FUNCTION_BLOCK FB_SDS
VAR_IN_OUT
    stSDS : ST_SDS;
    stSDSPersistent : ST_SDSPersistent;
END_VAR
VAR
    nIndex: UINT;

    fbStateSetup: FB_StateSetupHelper;
    stDefault: ST_PositionState := (
        fDelta := 0.5,
        fVelocity := 1,
        bMoveOk := TRUE,
        bValid := TRUE
    );
END_VAR


// Check the present homing status
ACT_CheckHomeStatus();

IF NOT stSDSPersistent.bInitialized THEN
    // Do all the required initialization for the persistent data of the sample delivery system.

    stSDSPersistent.stTransferArmSlot.sTag := 'TA';
    stSDSPersistent.stDiffractometerSlot.sTag := 'DF';

    FOR nIndex := E_SDSGarageYStates.T1 to E_SDSGarageYStates.B4 BY 1 DO
        stSDSPersistent.astGarageSlot[nIndex].eState := E_SampleSlotStates.EMPTY;
        stSDSPersistent.astGarageSlot[nIndex].sDesc  := '';
    END_FOR

    stSDSPersistent.astGarageSlot[E_SDSGarageYStates.T1].sTag := 'T1';

    stSDSPersistent.astGarageSlot[E_SDSGarageYStates.T1].fDeg := 0.0;
    stSDSPersistent.astGarageSlot[E_SDSGarageYStates.M1].fDeg := 0.0;
    stSDSPersistent.astGarageSlot[E_SDSGarageYStates.B1].fDeg := 0.0;

    stSDSPersistent.astGarageSlot[E_SDSGarageYStates.T2].fDeg := 90.0;
    stSDSPersistent.astGarageSlot[E_SDSGarageYStates.M2].fDeg := 90.0;
    stSDSPersistent.astGarageSlot[E_SDSGarageYStates.B2].fDeg := 90.0;

    stSDSPersistent.astGarageSlot[E_SDSGarageYStates.T3].fDeg := 180.0;
    stSDSPersistent.astGarageSlot[E_SDSGarageYStates.M3].fDeg := 180.0;
    stSDSPersistent.astGarageSlot[E_SDSGarageYStates.B3].fDeg := 180.0;

    stSDSPersistent.astGarageSlot[E_SDSGarageYStates.T4].fDeg := 270.0;
    stSDSPersistent.astGarageSlot[E_SDSGarageYStates.M4].fDeg := 270.0;
    stSDSPersistent.astGarageSlot[E_SDSGarageYStates.B4].fDeg := 270.0;

    stSDSPersistent.astGarageSlot[E_SDSGarageYStates.T1].fYPos := -100.5;
    stSDSPersistent.astGarageSlot[E_SDSGarageYStates.T2].fYPos := -100.5;
    stSDSPersistent.astGarageSlot[E_SDSGarageYStates.T3].fYPos := -100.5;
    stSDSPersistent.astGarageSlot[E_SDSGarageYStates.T4].fYPos := -100.5;

    stSDSPersistent.astGarageSlot[E_SDSGarageYStates.M1].fYPos := -74.5;
    stSDSPersistent.astGarageSlot[E_SDSGarageYStates.M2].fYPos := -74.5;
    stSDSPersistent.astGarageSlot[E_SDSGarageYStates.M3].fYPos := -74.5;
    stSDSPersistent.astGarageSlot[E_SDSGarageYStates.M4].fYPos := -74.5;

    stSDSPersistent.astGarageSlot[E_SDSGarageYStates.B1].fYPos := -44.5;
    stSDSPersistent.astGarageSlot[E_SDSGarageYStates.B2].fYPos := -44.5;
    stSDSPersistent.astGarageSlot[E_SDSGarageYStates.B3].fYPos := -44.5;
    stSDSPersistent.astGarageSlot[E_SDSGarageYStates.B4].fYPos := -44.5;

    stSDSPersistent.fGarageHeightSafeFromCollision := -40.0;
    stSDSPersistent.fGarageRotationClearanceOffset := 45.0;

    stSDSPersistent.bInitialized := TRUE;
END_IF

IF NOT stSDS.bInitialized THEN
    // Do all the required initialization for the non-persistent data of the sample delivery system.
    stSDS.bHomingRequired := TRUE;

    fbStateSetup(stPositionState:=stDefault, bSetDefault:=TRUE);

    stSDS.bInitialized := TRUE;
END_IF

// Update load/unloadable statuses for the garage, transfer arm, and the diffractometer.
UpdateLoadUnloadAbleStatuses(
    stSDS := stSDS,
    stSDSP := stSDSPersistent
);

// Check if garage is above the threshold to rotate freely without fear of hitting the transfer arm.
ConfirmGarageFreeToRotate(
    stSDS := stSDS,
    stSDSP := stSDSPersistent
);

// Control the sequencing of the sample delivery system.
StateMachine(
    stSDS := stSDS,
    stSDSP := stSDSPersistent
);

// Update the position states
UpdatePositionStates(
    stSDS := stSDS,
    stSDSP := stSDSPersistent
);

// Call state position function blocks.
stSDS.fbTransferArmHPos1D(
    stMotionStage:=stSDS.stTransferArmHStage,
    astPositionState:=stSDS.astTransferArmHPosState,
    eEnumSet:=stSDS.eTransferArmHStateSet,
    eEnumGet:=stSDS.eTransferArmHStateGet,
    bEnable:=TRUE,
    stEpicsToPlc:=stSDS.stTransferArmHEpicsToPlc,
    stPlcToEpics=>stSDS.stTransferArmHPlcToEpics
);
stSDS.fbTransferArmRPos1D(
    stMotionStage:=stSDS.stTransferArmRStage,
    astPositionState:=stSDS.astTransferArmRPosState,
    eEnumSet:=stSDS.eTransferArmRStateSet,
    eEnumGet:=stSDS.eTransferArmRStateGet,
    bEnable:=TRUE,
    stEpicsToPlc:=stSDS.stTransferArmREpicsToPlc,
    stPlcToEpics=>stSDS.stTransferArmRPlcToEpics
);

stSDS.fbGarageYPos1D(
    stMotionStage:=stSDS.stGarageYStage,
    astPositionState:=stSDS.astGarageYPosState,
    eEnumSet:=stSDS.eGarageYStateSet,
    eEnumGet:=stSDS.eGarageYStateGet,
    bEnable:=TRUE,
    stEpicsToPlc:=stSDS.stGarageYEpicsToPlc,
    stPlcToEpics=>stSDS.stGarageYPlcToEpics
);

stSDS.fbGarageRPos1D(
    stMotionStage:=stSDS.stGarageRStage,
    astPositionState:=stSDS.astGarageRPosState,
    eEnumSet:=stSDS.eGarageRStateSet,
    eEnumGet:=stSDS.eGarageRStateGet,
    bEnable:=TRUE,
    stEpicsToPlc:=stSDS.stGarageREpicsToPlc,
    stPlcToEpics=>stSDS.stGarageRPlcToEpics
);

// Ensure UI boolean commands are cleared after holding for one second.
HoldThenClear(b1 := stSDS.stUISelect.bExitManualControl, tHoldDuration := T#1s);
HoldThenClear(b1 := stSDS.stUISelect.bHomeGarage, tHoldDuration := T#1s);
HoldThenClear(b1 := stSDS.stUISelect.bHomeTransferArm, tHoldDuration := T#1s);
HoldThenClear(b1 := stSDS.stUISelect.bLoad, tHoldDuration := T#1s);
HoldThenClear(b1 := stSDS.stUISelect.bLoadArmFromGarage, tHoldDuration := T#1s);
HoldThenClear(b1 := stSDS.stUISelect.bLoadDiffractometerFromArm, tHoldDuration := T#1s);
HoldThenClear(b1 := stSDS.stUISelect.bLoadGarageFromPort, tHoldDuration := T#1s);
HoldThenClear(b1 := stSDS.stUISelect.bLoadUnloadGarageFromPort, tHoldDuration := T#1s);
HoldThenClear(b1 := stSDS.stUISelect.bManualControl, tHoldDuration := T#1s);
HoldThenClear(b1 := stSDS.stUISelect.bProceed, tHoldDuration := T#1s);
HoldThenClear(b1 := stSDS.stUISelect.bUnload, tHoldDuration := T#1s);
HoldThenClear(b1 := stSDS.stUISelect.bUnloadArmToGarage, tHoldDuration := T#1s);
HoldThenClear(b1 := stSDS.stUISelect.bUnloadDiffractometerToArm, tHoldDuration := T#1s);

// Align with the saved selection at the end of each cycle.
stSDS.stUISelect.eGarageSlot := stSDS.eSelectedGarageSlot;

ACTION ACT_CheckHomeStatus:

// ACTION - Check home status

CASE stSDS.nHomingState OF
    0: // Initialization
        stSDS.tonForwardHomingLimit(IN:=FALSE);
        IF stSDS.stTransferArmHStage.nCommand = E_EpicsMotorCmd.HOME AND stSDS.stTransferArmHStage.bBusy THEN
            stSDS.nHomingState := stSDS.nHomingState + 1;
        END_IF
    1: // Homing Sequence Triggered
        stSDS.tonForwardHomingLimit(IN:=stSDS.stTransferArmHStage.Axis.NcToPlc.SetVelo > 0,PT:=T#1s);
        IF stSDS.stTransferArmHStage.nCommand = E_EpicsMotorCmd.HOME AND stSDS.stTransferArmHStage.bHome THEN
            stSDS.nHomingState := stSDS.nHomingState + 1;
            stSDS.tonHomingStateTimeout(IN:=FALSE);
            stSDS.tonForwardHomingLimit(IN:=FALSE);
        ELSIF NOT stSDS.stTransferArmHStage.bBusy THEN
            stSDS.tonHomingStateTimeout(IN:=TRUE,PT:=T#5s);
            stSDS.tonForwardHomingLimit(IN:=FALSE);
            IF stSDS.tonHomingStateTimeout.Q THEN
                stSDS.nHomingState := -1;
            END_IF
        END_IF
    2: // Homing Sequence Successful
        IF F_Limit(stSDS.stTransferArmHStage.stAxisStatus.fActPosition, stSDS.stTransferArmHStage.fHomePosition-0.1, stSDS.stTransferArmHStage.fHomePosition+0.1, TRUE) THEN
            stSDS.bHomingRequired := FALSE;
            stSDS.nHomingState := 0;
            stSDS.tonHomingRequiredTimeout(IN:=FALSE);
            stSDS.tonHomingStateTimeout(IN:=FALSE);
        ELSIF NOT stSDS.stTransferArmHStage.bBusy THEN
            stSDS.tonHomingStateTimeout(IN:=TRUE,PT:=T#5s);
            IF stSDS.tonHomingStateTimeout.Q THEN
                stSDS.nHomingState := -1;
            END_IF
        END_IF
    -1: // Error Handling
        stSDS.nHomingState := 0;
END_CASE

stSDS.tonHomingRequiredTimeout(IN:=NOT stSDS.bHomingRequired,PT:=stSDS.tHomingRequiredTimeoutTime);
IF stSDS.tonHomingRequiredTimeout.Q THEN
    stSDS.bHomingRequired := TRUE;
END_IF
stSDS.fMinUntilHomingRequired := TIME_TO_REAL(stSDS.tonHomingRequiredTimeout.PT - stSDS.tonHomingRequiredTimeout.ET) / 60000;

IF stSDS.stTransferArmHStage.bExecute AND stSDS.bHomingRequired AND stSDS.stTransferArmHStage.fPosition > stSDS.stTransferArmHStage.stAxisStatus.fActPosition AND
    stSDS.stTransferArmHStage.nCommand <> E_EpicsMotorCmd.HOME THEN

    stSDS.stTransferArmHStage.bError := TRUE;
    stSDS.stTransferArmHStage.sCustomErrorMessage := 'Axis homing status overdue. Please home the axis.';
END_IF
END_ACTION


METHOD PRIVATE CheckCanDo2Criteria
VAR_IN_OUT
    bCanDo : BOOL;
    bCantDo : BOOL;
    sErrorMsg : T_MaxString;
END_VAR
VAR_INPUT
    b1 : BOOL;
    b2 : BOOL;
    sErrorMsgTF : T_MaxString;
    sErrorMsgFT : T_MaxString;
    sErrorMsgFF : T_MaxString;
END_VAR

bCanDo := FALSE;

IF b1 AND b2 THEN
    bCanDo := TRUE;
ELSIF b1 AND NOT b2 THEN
    bCantDo := TRUE;
    sErrorMsg := sErrorMsgTF;
ELSIF NOT b1 AND b2 THEN
    bCantDo := TRUE;
    sErrorMsg := sErrorMsgFT ;
ELSE
    bCantDo := TRUE;
    sErrorMsg := sErrorMsgFF;
END_IF
END_METHOD


METHOD PRIVATE CheckCanLoadArmFromGarage
VAR_IN_OUT
    stSDS : ST_SDS;
    stSDSP : ST_SDSPersistent;
END_VAR

stSDS.sStatusMsg := 'Checking if there is an open slot in the transfer arm and at least one full slot in the garage.';

CheckCanDo2Criteria(
    bCanDo := stSDS.bSuccess,
    bCantDo := stSDS.bError,
    sErrorMsg := stSDS.sErrorMsg,
    b1 := stSDS.bGarageUnloadable,
    b2 := stSDS.bTransferArmLoadable,
    sErrorMsgTF := 'The transfer arm is currently full and cannot be used to remove a sample from the garage.',
    sErrorMsgFT := 'The garage is currently empty and therefore no samples can be removed.',
    sErrorMsgFF := 'The garage is currently empty and the transfer arm is full. Therefore, no samples can be removed.'
);
END_METHOD


METHOD PRIVATE CheckCanLoadDiffractometerFromArm
VAR_IN_OUT
    stSDS : ST_SDS;
    stSDSP : ST_SDSPersistent;
END_VAR

stSDS.sStatusMsg := 'Checking if the diffractometer slot is open and if the transfer arm is carrying a sample.';

CheckCanDo2Criteria(
    bCanDo := stSDS.bSuccess,
    bCantDo := stSDS.bError,
    sErrorMsg := stSDS.sErrorMsg,
    b1 := stSDS.bDiffractometerLoadable,
    b2 := stSDS.bTransferArmUnloadable,
    sErrorMsgTF := 'The transfer arm is currently empty and cannot be used to place a sample in the diffractometer.',
    sErrorMsgFT := 'The diffractometer already has a sample in it.',
    sErrorMsgFF := 'The diffractoemter already has a sample and the transfer arm is empty.'
);
END_METHOD


METHOD PRIVATE CheckCanLoadUnloadGarageFromPort
VAR_IN_OUT
    stSDS : ST_SDS;
    stSDSP : ST_SDSPersistent;
END_VAR

stSDS.sStatusMsg := 'Checking if the garage can be loaded or unloaded from the port.';

stSDS.bSuccess := TRUE;
END_METHOD


METHOD PRIVATE CheckCanUnloadArmToGarage
VAR_IN_OUT
    stSDS : ST_SDS;
    stSDSP : ST_SDSPersistent;
END_VAR

stSDS.sStatusMsg := 'Checking if there is an open slot in the garage and if the transfer arm is carrying a sample.';

CheckCanDo2Criteria(
    bCanDo := stSDS.bSuccess,
    bCantDo := stSDS.bError,
    sErrorMsg := stSDS.sErrorMsg,
    b1 := stSDS.bGarageLoadable,
    b2 := stSDS.bTransferArmUnloadable,
    sErrorMsgTF := 'The transfer arm is currently empty and cannot be used to load sample into the garage.',
    sErrorMsgFT := 'The garage is currently full and therefore no samples can be loaded into it.',
    sErrorMsgFF := 'The garage is currently full and the transfer arm is empty.'
);
END_METHOD


METHOD PRIVATE CheckCanUnloadDiffractometerToArm
VAR_IN_OUT
    stSDS : ST_SDS;
    stSDSP : ST_SDSPersistent;
END_VAR

stSDS.sStatusMsg := 'Checking if the diffractometer slot is full and if the transfer arm is empty.';

CheckCanDo2Criteria(
    bCanDo := stSDS.bSuccess,
    bCantDo := stSDS.bError,
    sErrorMsg := stSDS.sErrorMsg,
    b1 := stSDS.bDiffractometerUnloadable,
    b2 := stSDS.bTransferArmLoadable,
    sErrorMsgTF := 'The transfer arm is currently full and cannot be used to unload a sample from the diffractometer.',
    sErrorMsgFT := 'The diffractometer does not have a sample in it.',
    sErrorMsgFF := 'The diffractometeris empty and the transfer arm is full.'
);
END_METHOD


METHOD PRIVATE ConfirmExtraction
VAR_IN_OUT
    stSDS : ST_SDS;
END_VAR

stSDS.bSuccess := FALSE;

stSDS.sStatusMsg := 'Moving transfer arm back a few mm. Please confirm the sample is held by the arm and then click "proceed". If the sample is still in the holder, click "retry" to go back to fine adjustment.';

SetPositionStateWaitForArrivalQuitIfError(
    eStateGet := stSDS.eTransferArmHStateGet,
    stMotionStage := stSDS.stTransferArmHStage,
    eStateSet := stSDS.eTransferArmHStateSet,
    eEnumSet := E_SDSTransferArmHStates.CONFIRM_GARAGE_EXTRACTION,
    bError := stSDS.bError,
    sErrorMsg := stSDS.sErrorMsg,
    bArrived => stSDS.bSuccess
);
END_METHOD


METHOD PRIVATE ConfirmGarageFreeToRotate
VAR_IN_OUT
    stSDS : ST_SDS;
    stSDSP : ST_SDSPersistent;
END_VAR

stSDS.bGarageAboveCollisionHeight := stSDS.stGarageYStage.Axis.NcToPlc.ActPos <= stSDSP.fGarageHeightSafeFromCollision;
END_METHOD


METHOD PRIVATE ConfirmInsertion
VAR_IN_OUT
    stSDS : ST_SDS;
END_VAR

stSDS.bSuccess := FALSE;

stSDS.sStatusMsg := 'Moving transfer arm back a few mm. Please confirm the sample is held by the garage and then click "proceed". If the sample is still in the transfer arm, click "retry" to go back to fine adjustment.';

SetPositionStateWaitForArrivalQuitIfError(
    eStateGet := stSDS.eTransferArmHStateGet,
    stMotionStage := stSDS.stTransferArmHStage,
    eStateSet := stSDS.eTransferArmHStateSet,
    eEnumSet := E_SDSTransferArmHStates.CONFIRM_GARAGE_INSERTION,
    bError := stSDS.bError,
    sErrorMsg := stSDS.sErrorMsg,
    bArrived => stSDS.bSuccess
);
END_METHOD


METHOD PRIVATE ConfirmSampleLoaded
VAR_INPUT
END_VAR
END_METHOD


METHOD PRIVATE ConfirmSampleUnloaded
VAR_INPUT
END_VAR
END_METHOD


METHOD PRIVATE ExtendPrerotateTransferArmForExtraction
VAR_IN_OUT
    stSDS : ST_SDS;
END_VAR
VAR
    bHArrived : BOOL;
    bRArrived : BOOL;
END_VAR

stSDS.bSuccess := FALSE;

stSDS.sStatusMsg := 'Moving transfer arm to nominal sample extraction position and pre-rotating to allow full rotation for unscrewing sample.';

SetPositionStateWaitForArrivalQuitIfError(
    eStateGet := stSDS.eTransferArmHStateGet,
    stMotionStage := stSDS.stTransferArmHStage,
    eStateSet := stSDS.eTransferArmHStateSet,
    eEnumSet := E_SDSTransferArmHStates.GARAGE_SAMPLE_REMOVAL,
    bError := stSDS.bError,
    sErrorMsg := stSDS.sErrorMsg,
    bArrived => bHArrived
);

SetPositionStateWaitForArrivalQuitIfError(
    eStateGet := stSDS.eTransferArmRStateGet,
    stMotionStage := stSDS.stTransferArmRStage,
    eStateSet := stSDS.eTransferArmRStateSet,
    eEnumSet := E_SDSTransferArmRStates.PREROTATE_SAMPLE_REMOVAL,
    bError := stSDS.bError,
    sErrorMsg := stSDS.sErrorMsg,
    bArrived => bRArrived
);

IF bHArrived AND bRArrived THEN
    stSDS.bSuccess := TRUE;
END_IF
END_METHOD


METHOD PRIVATE ExtendPrerotateTransferArmForLoading
VAR_IN_OUT
    stSDS : ST_SDS;
END_VAR
VAR
    bHArrived : BOOL;
    bRArrived : BOOL;
END_VAR

stSDS.bSuccess := FALSE;

stSDS.sStatusMsg := 'Moving transfer arm to nominal sample loading position and pre-rotating to allow full rotation for screwing in sample.';

SetPositionStateWaitForArrivalQuitIfError(
    eStateGet := stSDS.eTransferArmHStateGet,
    stMotionStage := stSDS.stTransferArmHStage,
    eStateSet := stSDS.eTransferArmHStateSet,
    eEnumSet := E_SDSTransferArmHStates.GARAGE_SAMPLE_INSERTION,
    bError := stSDS.bError,
    sErrorMsg := stSDS.sErrorMsg,
    bArrived => bHArrived
);

SetPositionStateWaitForArrivalQuitIfError(
    eStateGet := stSDS.eTransferArmRStateGet,
    stMotionStage := stSDS.stTransferArmRStage,
    eStateSet := stSDS.eTransferArmRStateSet,
    eEnumSet := E_SDSTransferArmRStates.PREROTATE_SAMPLE_INSERTION,
    bError := stSDS.bError,
    sErrorMsg := stSDS.sErrorMsg,
    bArrived => bRArrived
);

IF bHArrived AND bRArrived THEN
    stSDS.bSuccess := TRUE;
END_IF
END_METHOD


METHOD PRIVATE FineAdjustment
VAR_INPUT
END_VAR

stSDS.sStatusMsg := 'Use the individual motor control to do fine adjustment. Click "proceed" to move to the next step.';
END_METHOD


METHOD PRIVATE HoldThenClear
VAR_IN_OUT
    b1 : BOOL;
END_VAR
VAR_INPUT
    tHoldDuration : TIME := T#1s;
END_VAR
VAR_INST
    tonHoldTimer : TON;
END_VAR

tonHoldTimer(IN := b1, PT := tHoldDuration);

IF tonHoldTimer.Q THEN
    b1 := FALSE;
END_IF
END_METHOD


METHOD PRIVATE HomeGarage
VAR_INPUT
    stSDS : ST_SDS;
END_VAR

stSDS.bSuccess := FALSE;

stSDS.sStatusMsg := 'Homing the garage.';

IF stSDS.stGarageRStage.bError THEN
    stSDS.bError := TRUE;
    stSDS.sErrorMsg := 'Garage rotational stage has an active error. Aborting sequence.';
END_IF

HomeStateMachine(
    eHomingState := stSDS.eGarageRHomingState,
    stMotionStage := stSDS.stGarageRStage,
    bError => stSDS.bError,
    sErrorMsg => stSDS.sErrorMsg
);

IF stSDS.eGarageRHomingState = E_SDSHomingState.HOMED THEN
    stSDS.bSuccess := TRUE;
END_IF
END_METHOD


METHOD PRIVATE HomeStateMachine
VAR_IN_OUT
    eHomingState : E_SDSHomingState;
    stMotionStage : ST_MotionStage;
END_VAR
VAR_OUTPUT
    bError : BOOL;
    sErrorMsg : T_MaxString;
END_VAR

CASE eHomingState OF
    E_SDSHomingState.INIT:
        eHomingState := E_SDSHomingState.WAIT_NOT_BUSY;
    E_SDSHomingState.WAIT_NOT_BUSY:
        IF NOT stMotionStage.bBusy THEN
            eHomingState := E_SDSHomingState.TRIGGER_HOMING;
        END_IF
    E_SDSHomingState.TRIGGER_HOMING:
        stMotionStage.bHomeCmd := TRUE;
        IF stMotionStage.nCommand = E_EpicsMotorCmd.HOME AND stMotionStage.bBusy THEN
            eHomingState := E_SDSHomingState.WAIT_FOR_HOMED;
        END_IF
    E_SDSHomingState.WAIT_FOR_HOMED:
        IF stMotionStage.bDone THEN
            eHomingState := E_SDSHomingState.HOMED;
        END_IF
ELSE
    bError := TRUE;
    sErrorMsg := 'Homing sequence triggered an unknown state. Aborting sequence.';
END_CASE
END_METHOD


METHOD PRIVATE HomeTransferArm
VAR_IN_OUT
    stSDS : ST_SDS;
END_VAR

stSDS.bSuccess := FALSE;

stSDS.sStatusMsg := 'Homing the transfer arm.';

IF stSDS.stTransferArmHStage.bError THEN
    stSDS.bError := TRUE;
    stSDS.sErrorMsg := 'Transfer arm horizontal stage has an active error. Aborting sequence.';
END_IF

IF stSDS.stTransferArmRStage.bError THEN
    stSDS.bError := TRUE;
    stSDS.sErrorMsg := 'Transfer arm rotational stage has an active error. Aborting sequence.';
END_IF

HomeStateMachine(
    eHomingState := stSDS.eTransferArmHHomingState,
    stMotionStage := stSDS.stTransferArmHStage,
    bError => stSDS.bError,
    sErrorMsg => stSDS.sErrorMsg
);

HomeStateMachine(
    eHomingState := stSDS.eTransferArmRHomingState,
    stMotionStage := stSDS.stTransferArmRStage,
    bError => stSDS.bError,
    sErrorMsg => stSDS.sErrorMsg
);

IF stSDS.eTransferArmHHomingState = E_SDSHomingState.HOMED AND
   stSDS.eTransferArmRHomingState = E_SDSHomingState.HOMED THEN
    stSDS.bSuccess := TRUE;
END_IF
END_METHOD


METHOD PRIVATE InitHomeGarage
VAR_IN_OUT
    stSDS : ST_SDS;
END_VAR

stSDS.eGarageRHomingState := E_SDSHomingState.INIT;
END_METHOD


METHOD PRIVATE InitHomeTransferArm
VAR_IN_OUT
    stSDS : ST_SDS;
END_VAR

stSDS.eTransferArmHHomingState := E_SDSHomingState.INIT;
stSDS.eTransferArmRHomingState := E_SDSHomingState.INIT;
END_METHOD


METHOD PRIVATE InitRotateGarageForClearance
VAR_IN_OUT
    stSDS : ST_SDS;
    stSDSP : ST_SDSPersistent;
END_VAR

stSDS.fGarageRotationClearancePos := stSDS.stGarageRStage.Axis.NcToPlc.ActPos + stSDSP.fGarageRotationClearanceOffset;
END_METHOD


METHOD PRIVATE InitSelectGarageSlotForLoading
VAR_IN_OUT
    stSDS : ST_SDS;
    stSDSP : ST_SDSPersistent;
END_VAR

FOR nIndex := E_SDSGarageYStates.T1 TO E_SDSGarageYStates.B4 BY 1 DO
    CASE stSDSP.astGarageSlot[nIndex].eState OF
        E_SampleSlotStates.EMPTY:
            stSDS.eSelectedGarageSlot := nIndex;
    END_CASE
END_FOR

IF nIndex > E_SDSGarageYStates.B4 THEN
    stSDS.bError := TRUE;
    stSDS.sErrorMsg := 'There are no empty slots in the garage to load a sample to.';
END_IF
END_METHOD


METHOD PRIVATE InitSelectGarageSlotForRemoval
VAR_IN_OUT
    stSDS : ST_SDS;
    stSDSP : ST_SDSPersistent;
END_VAR

FOR nIndex := E_SDSGarageYStates.T1 TO E_SDSGarageYStates.B4 BY 1 DO
    CASE stSDSP.astGarageSlot[nIndex].eState OF
        E_SampleSlotStates.FULL:
            stSDS.eSelectedGarageSlot := nIndex;
    END_CASE
END_FOR

IF nIndex > E_SDSGarageYStates.B4 THEN
    stSDS.bError := TRUE;
    stSDS.sErrorMsg := 'There are no full slots in the garage to extract a sample from.';
END_IF
END_METHOD


METHOD PRIVATE ManualControl
VAR_INPUT
    stSDS : ST_SDS;
END_VAR
END_METHOD


METHOD PRIVATE MoveToGarageSlotFaceTransferArm
VAR_IN_OUT
    stSDS : ST_SDS;
END_VAR
VAR
    bYArrived : BOOL;
    bRArrived : BOOL;
END_VAR

stSDS.bSuccess := FALSE;

stSDS.sStatusMsg := 'Moving garage to selected slot and facing it towards transfer arm.';

stSDS.eFaceState := E_SDSFaceState.FACE_TRANSFER_ARM;

SetPositionStateWaitForArrivalQuitIfError(
    eStateGet := stSDS.eGarageYStateGet,
    stMotionStage := stSDS.stGarageYStage,
    eStateSet := stSDS.eGarageYStateSet,
    eEnumSet := stSDS.eSelectedGarageSlot,
    bError := stSDS.bError,
    sErrorMsg := stSDS.sErrorMsg,
    bArrived => bYArrived
);

SetPositionStateWaitForArrivalQuitIfError(
    eStateGet := stSDS.eGarageRStateGet,
    stMotionStage := stSDS.stGarageRStage,
    eStateSet := stSDS.eGarageRStateSet,
    eEnumSet := stSDS.eSelectedGarageSlot,
    bError := stSDS.bError,
    sErrorMsg := stSDS.sErrorMsg,
    bArrived => bRArrived
);

IF bYArrived AND bRArrived THEN
    stSDS.bSuccess := TRUE;
END_IF
END_METHOD


METHOD PRIVATE MoveToGarageSlotHeight
VAR_IN_OUT
    stSDS : ST_SDS;
END_VAR

stSDS.bSuccess := FALSE;

stSDS.sStatusMsg := 'Moving garage to selected slot height.';

SetPositionStateWaitForArrivalQuitIfError(
    eStateGet := stSDS.eGarageYStateGet,
    stMotionStage := stSDS.stGarageYStage,
    eStateSet := stSDS.eGarageYStateSet,
    eEnumSet := stSDS.eSelectedGarageSlot,
    bError := stSDS.bError,
    sErrorMsg := stSDS.sErrorMsg,
    bArrived => stSDS.bSuccess
);
END_METHOD


METHOD PRIVATE RetractGarage
VAR_IN_OUT
    stSDS : ST_SDS;
END_VAR

stSDS.bSuccess := FALSE;

stSDS.sStatusMsg := 'Retracting garage.';

SetPositionStateWaitForArrivalQuitIfError(
    eStateGet := stSDS.eGarageYStateGet,
    stMotionStage := stSDS.stGarageYStage,
    eStateSet := stSDS.eGarageYStateSet,
    eEnumSet := E_SDSGarageYStates.RETRACTED,
    bError := stSDS.bError,
    sErrorMsg := stSDS.sErrorMsg,
    bArrived => stSDS.bSuccess
);
END_METHOD


METHOD PRIVATE RotateGarageForClearance
VAR_IN_OUT
    stSDS : ST_SDS;
END_VAR

stSDS.bSuccess := FALSE;

stSDS.sStatusMsg := 'Rotating garage to prevent a collision with the transfer arm sample during movement of the garage.';

IF F_Limit(
       fVal := stSDS.stGarageRStage.Axis.NcToPlc.ActPos,
       fLLim := stSDS.fGarageRotationClearancePos - stSDS.stGarageRStage.stAxisParameters.fTargetPosControlRange,
       fHLim := stSDS.fGarageRotationClearancePos + stSDS.stGarageRStage.stAxisParameters.fTargetPosControlRange,
       bInclusive := FALSE
   ) AND NOT stSDS.stGarageRStage.bBusy THEN
   stSDS.bSuccess := TRUE;
ELSE
    stSDS.stGarageRStage.fPosition := stSDS.fGarageRotationClearancePos;
    stSDS.stGarageRStage.fVelocity := stSDS.fGarageRotationSpeed;
    stSDS.stGarageRStage.bMoveCmd := TRUE;
END_IF
END_METHOD


METHOD PRIVATE RotateGarageForClearanceManual
VAR_IN_OUT
    stSDS : ST_SDS;
END_VAR

stSDS.sStatusMsg := 'Please manually rotate the garage to 45 degrees, to prevent it from colliding with the sample on the transfer arm when raising it up. Click "proceed" when complete.';
END_METHOD


METHOD PRIVATE RotateToFacePort
VAR_IN_OUT
    stSDS : ST_SDS;
END_VAR

stSDS.bSuccess := FALSE;

stSDS.sStatusMsg := 'Rotating garage so that the selected slot faces the side port.';

stSDS.eFaceState := E_SDSFaceState.FACE_SIDE_PORT;

SetPositionStateWaitForArrivalQuitIfError(
    eStateGet := stSDS.eGarageRStateGet,
    stMotionStage := stSDS.stGarageRStage,
    eStateSet := stSDS.eGarageRStateSet,
    eEnumSet := stSDS.eSelectedGarageSlot,
    bError := stSDS.bError,
    sErrorMsg := stSDS.sErrorMsg,
    bArrived => stSDS.bSuccess
);
END_METHOD


METHOD PRIVATE RotateToFaceTransferArm
VAR_IN_OUT
    stSDS : ST_SDS;
END_VAR

stSDS.bSuccess := FALSE;

stSDS.sStatusMsg := 'Rotating garage so that the selected slot faces the transfer arm.';

stSDS.eFaceState := E_SDSFaceState.FACE_TRANSFER_ARM;

SetPositionStateWaitForArrivalQuitIfError(
    eStateGet := stSDS.eGarageRStateGet,
    stMotionStage := stSDS.stGarageRStage,
    eStateSet := stSDS.eGarageRStateSet,
    eEnumSet := stSDS.eSelectedGarageSlot,
    bError := stSDS.bError,
    sErrorMsg := stSDS.sErrorMsg,
    bArrived => stSDS.bSuccess
);
END_METHOD


METHOD PRIVATE ScrewSampleIntoGarage
VAR_IN_OUT
    stSDS : ST_SDS;
END_VAR

stSDS.bSuccess := FALSE;

stSDS.sStatusMsg := 'Screwing sample into garage. Click "proceed" when complete. To go back and retry fine adjustment, click "retry".';

SetPositionStateWaitForArrivalQuitIfError(
    eStateGet := stSDS.eTransferArmRStateGet,
    stMotionStage := stSDS.stTransferArmRStage,
    eStateSet := stSDS.eTransferArmRStateSet,
    eEnumSet := E_SDSTransferArmRStates.SCREW_INTO_GARAGE,
    bError := stSDS.bError,
    sErrorMsg := stSDS.sErrorMsg,
    bArrived => stSDS.bSuccess
);
END_METHOD


METHOD PRIVATE SelectDesiredAction
VAR_INPUT
    stSDS : ST_SDS;
END_VAR

stSDS.sStatusMsg := 'Please select the desired action.';
END_METHOD


METHOD PRIVATE SelectGarageSlotForLoading
VAR_IN_OUT
    stSDS : ST_SDS;
    stSDSP : ST_SDSPersistent;
END_VAR

stSDS.sStatusMsg := 'Please select a valid garage slot to load a sample to and then click "proceed".';

IF stSDS.stUISelect.eGarageSlot >= E_SDSGarageYStates.T1 AND stSDS.stUISelect.eGarageSlot <= E_SDSGarageYStates.B4 THEN
    CASE stSDSP.astGarageSlot[stSDS.stUISelect.eGarageSlot].eState OF
        E_SampleSlotStates.DISABLED:
            stSDS.sErrorMsg := 'The selected garage slot is currently disabled.';
        E_SampleSlotStates.EMPTY:
            stSDS.eSelectedGarageSlot := stSDS.stUISelect.eGarageSlot;
        E_SampleSlotStates.FULL:
            stSDS.sErrorMsg := 'The selected garage slot is currently full.';
    END_CASE
ELSE
    stSDS.sErrorMsg := 'Please select a valid slot from T1 to B4.';
END_IF
END_METHOD


METHOD PRIVATE SelectGarageSlotForRemoval
VAR_IN_OUT
    stSDS : ST_SDS;
    stSDSP : ST_SDSPersistent;
END_VAR

stSDS.sStatusMsg := 'Please select a valid garage slot to retrieve a sample from and then click "proceed".';

IF stSDS.stUISelect.eGarageSlot >= E_SDSGarageYStates.T1 AND stSDS.stUISelect.eGarageSlot <= E_SDSGarageYStates.B4 THEN
    CASE stSDSP.astGarageSlot[stSDS.stUISelect.eGarageSlot].eState OF
        E_SampleSlotStates.DISABLED:
            stSDS.sErrorMsg := 'The selected garage slot is currently disabled.';
        E_SampleSlotStates.EMPTY:
            stSDS.sErrorMsg := 'The selected garage slot is currently empty.';
        E_SampleSlotStates.FULL:
            stSDS.eSelectedGarageSlot := stSDS.stUISelect.eGarageSlot;
    END_CASE
ELSE
    stSDS.sErrorMsg := 'Please select a valid slot from T1 to B4.';
END_IF
END_METHOD


METHOD PRIVATE SelectLoadUnloadGarage
VAR_IN_OUT
    stSDS : ST_SDS;
END_VAR

stSDS.sStatusMsg := 'Select whether you would like to load a sample to the garage or remove a sample to the garage.';

stSDS.bLoadingSelected := FALSE;
stSDS.bUnloadingSelected := FALSE;

IF stSDS.stUISelect.bLoad THEN
    stSDS.bLoadingSelected := TRUE;
ELSIF stSDS.stUISelect.bUnload THEN
    stSDS.bUnloadingSelected := TRUE;
END_IF
END_METHOD


METHOD PRIVATE SetPositionStateWaitForArrivalQuitIfError
VAR_IN_OUT
    eStateGet : UINT;
    stMotionStage : ST_MotionStage;
    eStateSet : UINT;
    bError : BOOL;
    sErrorMsg : T_MaxString;
END_VAR
VAR_INPUT
    eEnumSet : UINT;
END_VAR
VAR_OUTPUT
    bArrived : BOOL;
END_VAR

IF eStateGet = eEnumSet AND
    NOT stMotionStage.bBusy THEN
    bArrived := TRUE;
ELSIF stMotionStage.bError THEN
    bError := TRUE;
    sErrorMsg := 'And axis error occurred. Aborting sequence.';
END_IF

IF eStateGet <> eEnumSet THEN
    eStateSet := eEnumSet;
END_IF
END_METHOD


METHOD PRIVATE SetSeqState
VAR_INPUT
    stSDS : ST_SDS;
    eSeqState : E_SDSState;
END_VAR

stSDS.eSeqState := eSeqState;
END_METHOD


METHOD PRIVATE SetState
VAR_INPUT
    stSDS : ST_SDS;
    eState : E_SDSState;
END_VAR

stSDS.eState := eState;
END_METHOD


METHOD PRIVATE SetSubstate
VAR_INPUT
    stSDS : ST_SDS;
    eSubState : E_SDSState;
END_VAR

stSDS.eSubState := eSubState;
END_METHOD


METHOD PRIVATE StateMachine
VAR_IN_OUT
    stSDS : ST_SDS;
    stSDSP : ST_SDSPersistent;
END_VAR
END_METHOD


METHOD PRIVATE StateMachine_statechart
VAR_IN_OUT
    stSDS : ST_SDS;
    stSDSP : ST_SDSPersistent;
END_VAR
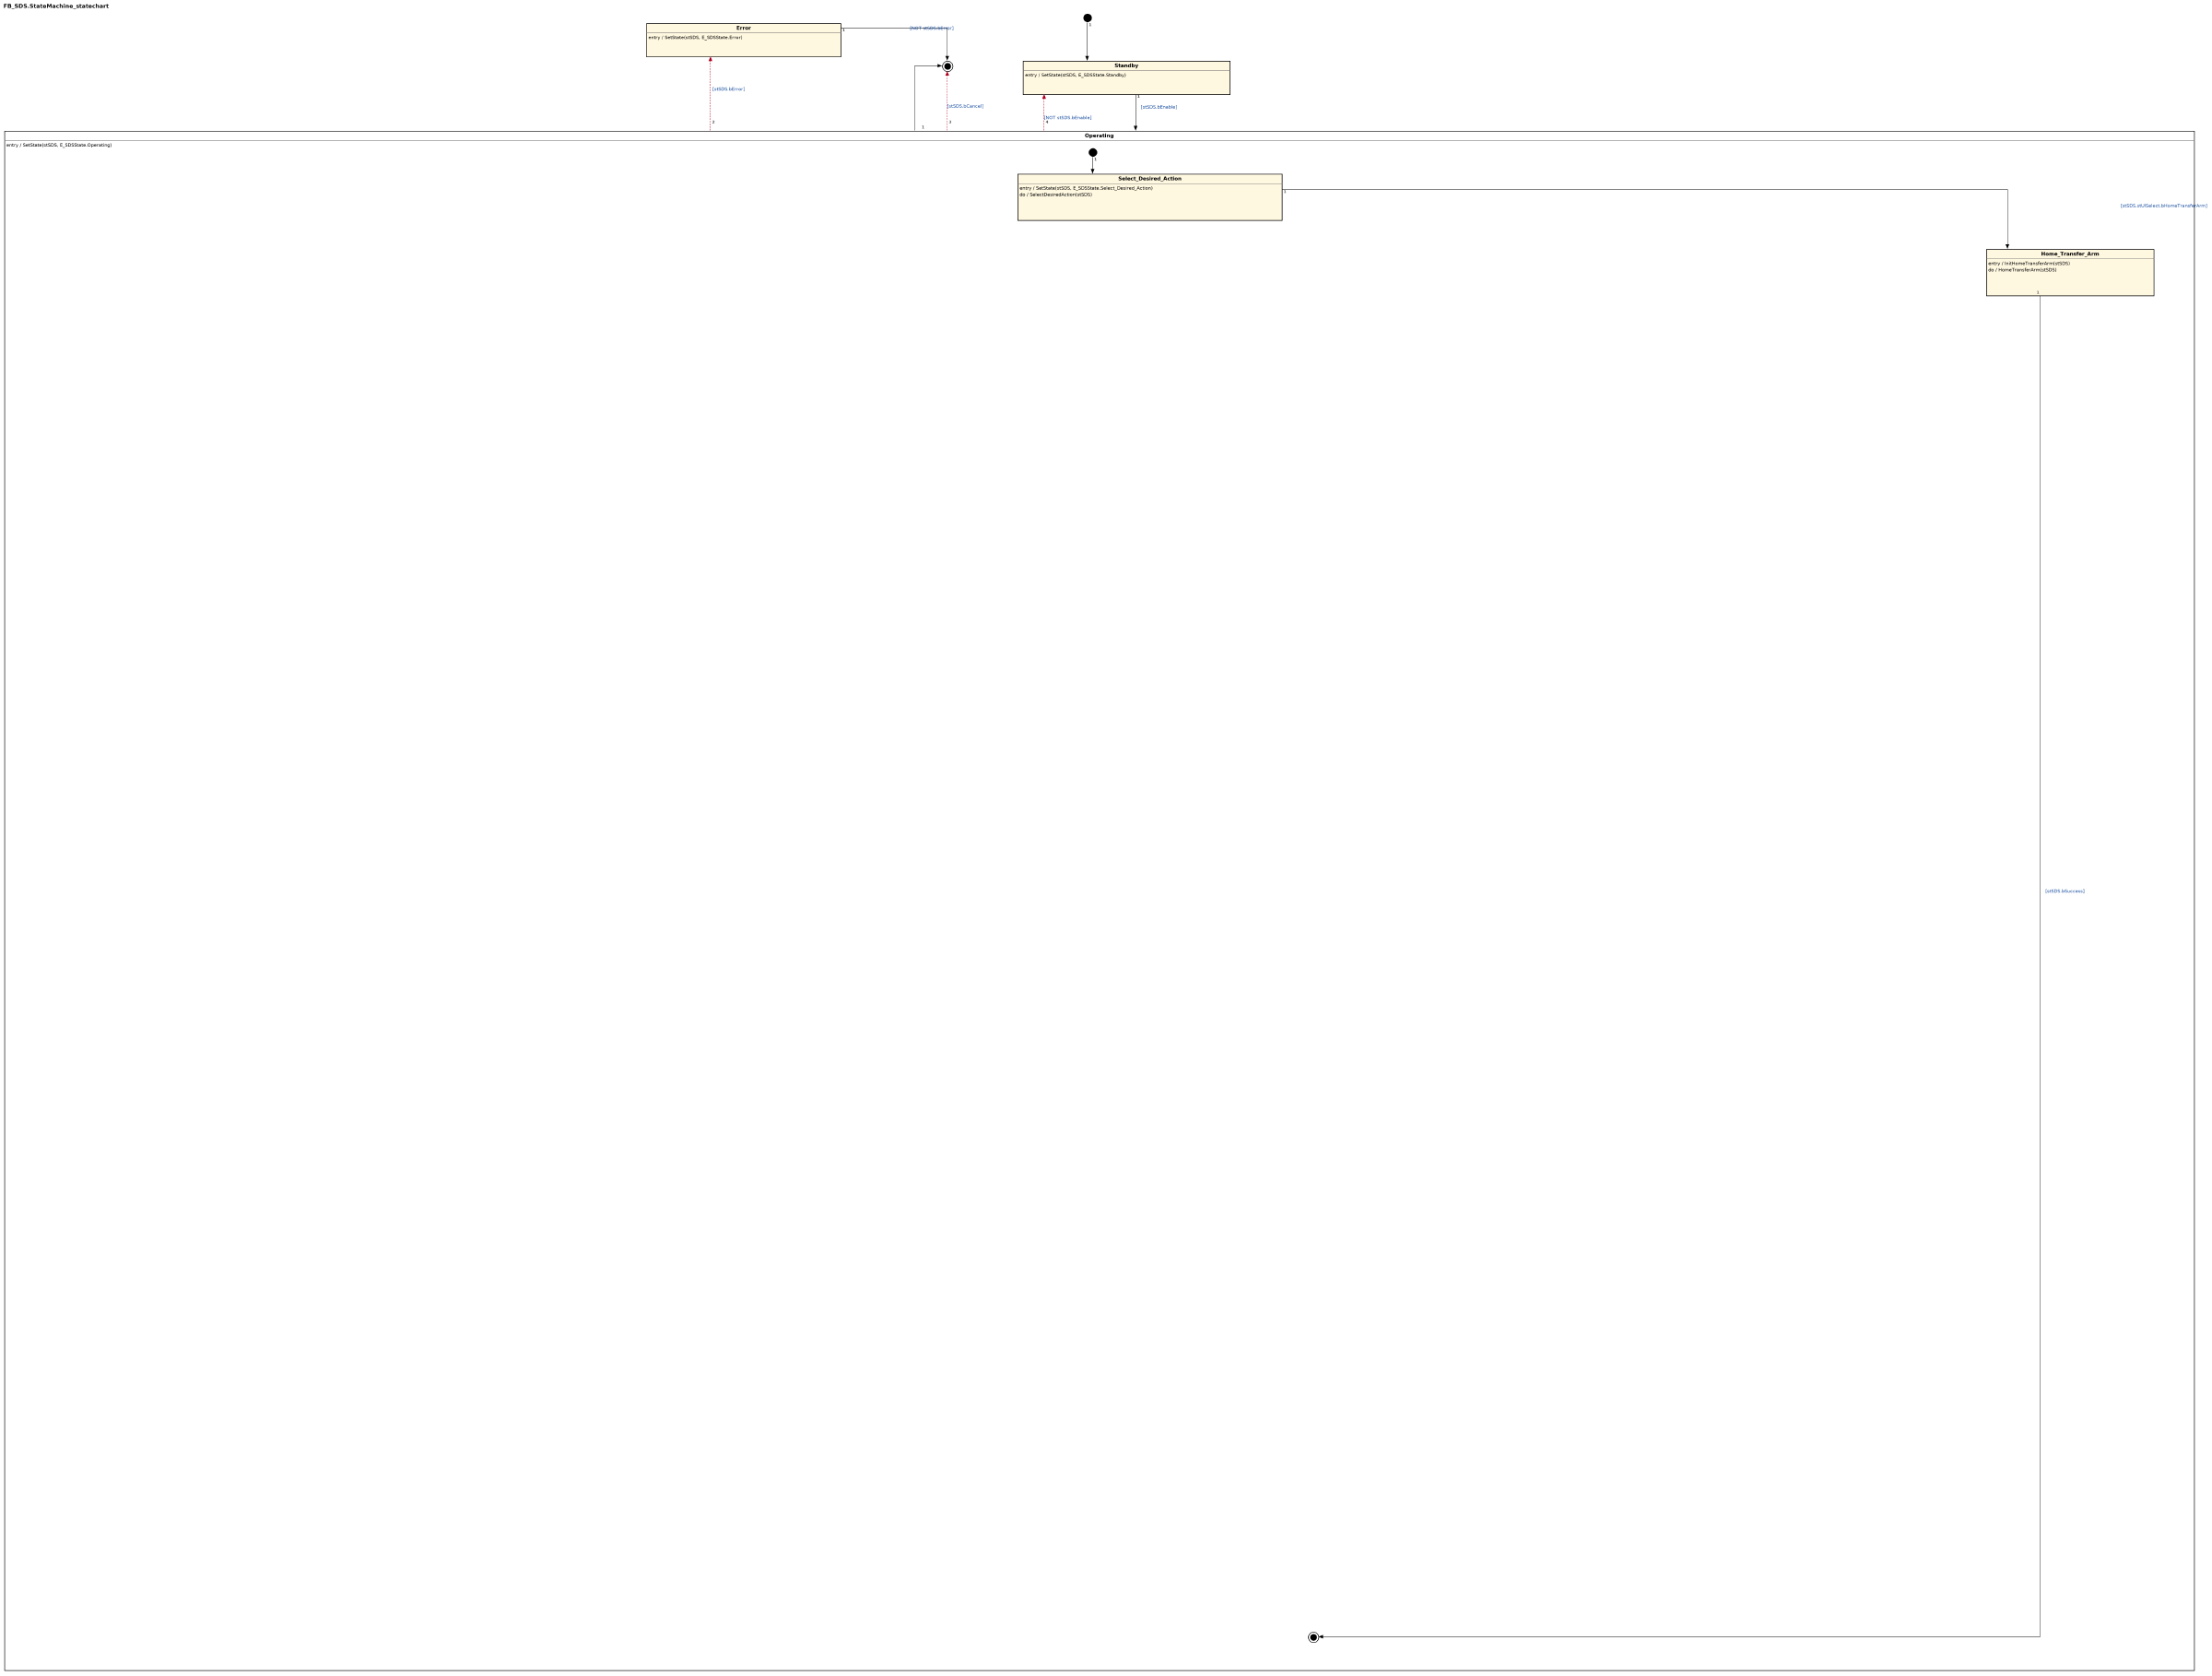
STATECHART StateMachine  // abortable
    START StartState1
    STATE Error
        entry / SetState(stSDS, E_SDSState.Error)
    END EndState3
    STATE Standby
        entry / SetState(stSDS, E_SDSState.Standby)
    COMPOSITE STATE Operating
        entry / SetState(stSDS, E_SDSState.Operating)
        START StartState1_copy_copy_copy_copy
        STATE Select_Desired_Action
            entry / SetState(stSDS, E_SDSState.Select_Desired_Action)
            do / SelectDesiredAction(stSDS)
        STATE Home_Transfer_Arm
            entry / InitHomeTransferArm(stSDS)
            do / HomeTransferArm(stSDS)
        END EndState2
        StartState1_copy_copy_copy_copy -> Select_Desired_Action  // priority 1, on completion
        Select_Desired_Action -> Home_Transfer_Arm [stSDS.stUISelect.bHomeTransferArm] // priority 1, rising edge
        Home_Transfer_Arm -> EndState2 [stSDS.bSuccess] // priority 1
    END_STATE
    StartState1 -> Standby  // priority 1, on completion
    Error -> EndState3 [NOT stSDS.bError] // priority 1
    Standby -> Operating [stSDS.bEnable] // priority 1
    Operating -> EndState3  // priority 1, on completion
    Operating -> Error [stSDS.bError] // priority 2, exception
    Operating -> EndState3 [stSDS.bCancel] // priority 3, exception
    Operating -> Standby [NOT stSDS.bEnable] // priority 4, exception
END_STATECHART
END_METHOD


METHOD PRIVATE UnscrewSampleFromGarage
VAR_IN_OUT
    stSDS : ST_SDS;
END_VAR

stSDS.bSuccess := FALSE;

stSDS.sStatusMsg := 'Unscrewing sample from garage. Click "proceed" when complete. To go back and retry fine adjustment, click "retry".';

SetPositionStateWaitForArrivalQuitIfError(
    eStateGet := stSDS.eTransferArmRStateGet,
    stMotionStage := stSDS.stTransferArmRStage,
    eStateSet := stSDS.eTransferArmRStateSet,
    eEnumSet := E_SDSTransferArmRStates.UNSCREW_FROM_GARAGE,
    bError := stSDS.bError,
    sErrorMsg := stSDS.sErrorMsg,
    bArrived => stSDS.bSuccess
);
END_METHOD


METHOD PRIVATE UpdateLoadUnloadAbleStatuses
VAR_IN_OUT
    stSDS : ST_SDS;
    stSDSP : ST_SDSPersistent;
END_VAR

// Determine whether the transfer arm is loadable or unloadable.
// If the transfer arm is disabled, then nothing is allowed.
// If the transfer arm is empty, it can be loaded.
// If the transfer arm is full, it can be unloaded.
CASE stSDSP.stTransferArmSlot.eState OF
    E_SampleSlotStates.EMPTY:
        stSDS.bTransferArmLoadable   := TRUE;
        stSDS.bTransferArmUnloadable := FALSE;
    E_SampleSlotStates.FULL:
        stSDS.bTransferArmLoadable   := FALSE;
        stSDS.bTransferArmUnloadable := TRUE;
    E_SampleSlotStates.DISABLED:
        stSDS.bTransferArmLoadable   := FALSE;
        stSDS.bTransferArmUnloadable := FALSE;
END_CASE

// Determine whether the diffractometer slot is loadable or unloadable.
// If the diffractometer slot is disabled, then nothing is allowed.
// If the diffractometer slot is empty, it can be loaded.
// If the diffractometer slot is full, it can be unloaded.
CASE stSDSP.stDiffractometerSlot.eState OF
    E_SampleSlotStates.EMPTY:
        stSDS.bDiffractometerLoadable   := TRUE;
        stSDS.bDiffractometerUnloadable := FALSE;
    E_SampleSlotStates.FULL:
        stSDS.bDiffractometerLoadable   := FALSE;
        stSDS.bDiffractometerUnloadable := TRUE;
    E_SampleSlotStates.DISABLED:
        stSDS.bDiffractometerLoadable   := FALSE;
        stSDS.bDiffractometerUnloadable := FALSE;
END_CASE

// Determine whether the garage is loadable or unloadable.
// If all slots in the garage are disabled, then nothing is allowed.
// If at least one slot in the garage is empty, it can be loaded.
// If at least one slot in the garage is full, it can be unloaded.
stSDS.bGarageLoadable := FALSE;
stSDS.bGarageUnloadable := FALSE;
FOR nIndex := 0 TO stSDS.nGarageSlots - 1 BY 1 DO
    CASE stSDSP.astGarageSlot[nIndex].eState OF
        E_SampleSlotStates.EMPTY:
            stSDS.bGarageLoadable   := TRUE;
        E_SampleSlotStates.FULL:
            stSDS.bGarageUnloadable := TRUE;
        E_SampleSlotStates.DISABLED:
            stSDS.bGarageLoadable := FALSE;
            stSDS.bGarageUnloadable := FALSE;
    END_CASE
END_FOR
END_METHOD


METHOD PRIVATE UpdatePositionStates
VAR_IN_OUT
    stSDS : ST_SDS;
    stSDSP : ST_SDSPersistent;
END_VAR

// Update parameters for transfer arm states.
// Horizontal axis states
fbStateSetup(stPositionState:=stSDS.astTransferArmHPosState[E_SDSTransferArmHStates.RETRACTED], sName:='RETRACTED',
    fPosition:=0,
    fVelocity:=2,
    fDelta := 2.5
);
fbStateSetup(stPositionState:=stSDS.astTransferArmHPosState[E_SDSTransferArmHStates.GARAGE_SAMPLE_REMOVAL], sName:='GARAGE_SAMPLE_REMOVAL',
    fPosition:=28,
    fVelocity:=2
);
fbStateSetup(stPositionState:=stSDS.astTransferArmHPosState[E_SDSTransferArmHStates.CONFIRM_GARAGE_EXTRACTION], sName:='CONFIRM_GARAGE_EXTRACTION',
    fPosition:=23,
    fVelocity:=2
);
fbStateSetup(stPositionState:=stSDS.astTransferArmHPosState[E_SDSTransferArmHStates.GARAGE_SAMPLE_INSERTION], sName:='GARAGE_SAMPLE_INSERTION',
    fPosition:=30,
    fVelocity:=2
);
fbStateSetup(stPositionState:=stSDS.astTransferArmHPosState[E_SDSTransferArmHStates.CONFIRM_GARAGE_INSERTION], sName:='CONFIRM_GARAGE_INSERTION',
    fPosition:=25,
    fVelocity:=2
);

// Rotational axis states
fbStateSetup(stPositionState:=stSDS.astTransferArmRPosState[E_SDSTransferArmRStates.FULLY_CCW], sName:='FULLY_CCW',
    fPosition:=0,
    fVelocity:=stSDS.fGarageRotationSpeed,
    fDelta := 5.0
);
fbStateSetup(stPositionState:=stSDS.astTransferArmRPosState[E_SDSTransferArmRStates.PREROTATE_SAMPLE_REMOVAL], sName:='PREROTATE_SAMPLE_REMOVAL',
    fPosition:=2000,
    fVelocity:=stSDS.fGarageRotationSpeed
);
fbStateSetup(stPositionState:=stSDS.astTransferArmRPosState[E_SDSTransferArmRStates.PREROTATE_SAMPLE_INSERTION], sName:='PREROTATE_SAMPLE_INSERTION',
    fPosition:=0,
    fVelocity:=stSDS.fGarageRotationSpeed
);
fbStateSetup(stPositionState:=stSDS.astTransferArmRPosState[E_SDSTransferArmRStates.UNSCREW_FROM_GARAGE], sName:='UNSCREW_FROM_GARAGE',
    fPosition:=0,
    fVelocity:=stSDS.fGarageRotationSpeed
);
fbStateSetup(stPositionState:=stSDS.astTransferArmRPosState[E_SDSTransferArmRStates.SCREW_INTO_GARAGE], sName:='SCREW_INTO_GARAGE',
    fPosition:=1700,
    fVelocity:=stSDS.fGarageRotationSpeed
);

// Update parameters for garage states.
// Y axis states
fbStateSetup(
    stPositionState := stSDS.astGarageYPosState[E_SDSGarageYStates.RETRACTED], sName:='RETRACTED',
    fPosition := 0.0,
    fVelocity := 2.0,
    fDelta := 10.0
);

FOR nIndex := E_SDSGarageYStates.T1 TO E_SDSGarageYStates.B4 BY 1 DO
    fbStateSetup(
        stPositionState := stSDS.astGarageYPosState[nIndex],
        sName := stSDSP.astGarageSlot[nIndex].sTag,
        fPosition := stSDSP.astGarageSlot[nIndex].fYPos,
        fVelocity := 2.0,
    );
END_FOR

// Rotational axis states
fbStateSetup(
    stPositionState := stSDS.astGarageRPosState[E_SDSGarageRStates.PREDICTED_HOME], sName:='PREDICTED_HOME',
    fPosition := 0.0,
    fVelocity := 10.0,
    fDelta := 1.0,
    bLocked := TRUE
);

FOR nIndex := E_SDSGarageYStates.T1 TO E_SDSGarageYStates.B4 BY 1 DO
    CASE stSDS.eFaceState OF
        E_SDSFaceState.FACE_SIDE_PORT:
            fbStateSetup(
                stPositionState := stSDS.astGarageRPosState[nIndex],
                sName := stSDSP.astGarageSlot[nIndex].sTag,
                fPosition := stSDSP.astGarageSlot[nIndex].fDeg + stSDS.fFacePortOffset,
                fVelocity := 10.0,
            );
    ELSE
        fbStateSetup(
            stPositionState := stSDS.astGarageRPosState[nIndex],
            sName := stSDSP.astGarageSlot[nIndex].sTag,
            fPosition := stSDSP.astGarageSlot[nIndex].fDeg,
            fVelocity := 10.0,
        );
    END_CASE
END_FOR
END_METHOD


METHOD PRIVATE UpdateSampleLocationDatabaseGarageToArm
VAR_IN_OUT
    stSDS : ST_SDS;
    stSDSP : ST_SDSPersistent;
END_VAR
VAR
    stTempSlot : ST_SampleSlot;
END_VAR

stSDS.bSuccess := FALSE;

stTempSlot := stSDSP.stTransferArmSlot;

stSDS.sStatusMsg := 'Updating the sample database.';

IF stSDS.eSelectedGarageSlot >= E_SDSGarageYStates.T1 AND stSDS.eSelectedGarageSlot <= E_SDSGarageYStates.B4 THEN
    stSDSP.stTransferArmSlot.eState := stSDSP.astGarageSlot[stSDS.eSelectedGarageSlot].eState;
    stSDSP.stTransferArmSlot.sDesc := stSDSP.astGarageSlot[stSDS.eSelectedGarageSlot].sDesc;

    stSDSP.astGarageSlot[stSDS.eSelectedGarageSlot].eState := stTempSlot.eState;
    stSDSP.astGarageSlot[stSDS.eSelectedGarageSlot].sDesc := stTempSlot.sDesc;

    stSDS.bSuccess := TRUE;
ELSE
    stSDS.sErrorMsg := 'Failed to automatically update sample position in database. Invalid slot selected. Sequence will continue, but please manually update the database from the interface. After manually updating the database, click "proceed" to continue.';
END_IF
END_METHOD


METHOD PRIVATE UpdateSampleLocationDatabaseManualExtraction
VAR_IN_OUT
    stSDS : ST_SDS;
    stSDSP : ST_SDSPersistent;
END_VAR

stSDS.bSuccess := FALSE;

stSDS.sStatusMsg := 'Please extract the sample. Click "proceed" when you have finished.';

IF stSDS.eSelectedGarageSlot >= E_SDSGarageYStates.T1 AND stSDS.eSelectedGarageSlot <= E_SDSGarageYStates.B4 THEN
    stSDSP.astGarageSlot[stSDS.eSelectedGarageSlot].eState := E_SampleSlotStates.EMPTY;
    stSDSP.astGarageSlot[stSDS.eSelectedGarageSlot].sDesc := '';
ELSE
    stSDS.sErrorMsg := 'Failed to update sample position in database. Invalid slot selected. Sequence will continue, but please manually update the database from the interface.';
END_IF
END_METHOD


METHOD PRIVATE UpdateSampleLocationDatabaseManualInsertion
VAR_IN_OUT
    stSDS : ST_SDS;
    stSDSP : ST_SDSPersistent;
END_VAR

stSDS.bSuccess := FALSE;

stSDS.sStatusMsg := 'Please insert the sample and write an identifying description for it in the text field. Click "proceed" when you have finished.';

IF stSDS.eSelectedGarageSlot >= E_SDSGarageYStates.T1 AND stSDS.eSelectedGarageSlot <= E_SDSGarageYStates.B4 THEN
    stSDSP.astGarageSlot[stSDS.eSelectedGarageSlot].eState := E_SampleSlotStates.FULL;
    stSDSP.astGarageSlot[stSDS.eSelectedGarageSlot].sDesc := stSDS.stUISelect.sTextInput;
ELSE
    stSDS.sErrorMsg := 'Failed to update sample position in database. Invalid slot selected. Sequence will continue, but please manually update the database from the interface.';
END_IF
END_METHOD

END_FUNCTION_BLOCK

(* stored: Version 1.1.0.1
   POU FB_SDS: Id {bf132679-4d4c-411f-a447-cbfc956c233d}, SpecialFunc None
   Action ACT_CheckHomeStatus: Id {2164ae39-f7d0-4dc9-a63c-01d4fb087899}
   Method CheckCanDo2Criteria: Id {0999b5e8-bb20-02f7-067b-9b396a45bac0}
   Method CheckCanLoadArmFromGarage: Id {d135d403-d5a2-0876-3e20-9dcee1c040ff}
   Method CheckCanLoadDiffractometerFromArm: Id {71a9fba2-1bcf-05b9-058e-f9891ff23ef5}
   Method CheckCanLoadUnloadGarageFromPort: Id {b5df68c0-c587-0d44-3d7f-12592aad6aff}
   Method CheckCanUnloadArmToGarage: Id {bb78d83b-b077-07a7-1d29-968f5b337faf}
   Method CheckCanUnloadDiffractometerToArm: Id {06a3e562-c435-024f-1e8f-6fea08c3c9bc}
   Method ConfirmExtraction: Id {daf24cc7-3887-03b2-0501-848224111e75}
   Method ConfirmGarageFreeToRotate: Id {80a711c4-d62e-03ac-2a4e-7a389529de7a}
   Method ConfirmInsertion: Id {5b3d04ea-c8d6-05a9-2354-558daca75a4d}
   Method ConfirmSampleLoaded: Id {59212a0a-1d84-0106-05ab-0993ad636ffe}
   Method ConfirmSampleUnloaded: Id {a0f2d941-1761-0fd5-2fd9-ad0713111335}
   Method ExtendPrerotateTransferArmForExtraction: Id {571dc7b2-1f9e-05ae-158e-96ba0d810ede}
   Method ExtendPrerotateTransferArmForLoading: Id {b432a359-f29f-08b6-14e5-baa64277214a}
   Method FineAdjustment: Id {51bb2359-fcd7-0761-04cb-c7da836e46a0}
   Method HoldThenClear: Id {c1475491-9357-0fa0-082d-566521e8e794}
   Method HomeGarage: Id {e7f9863f-7463-0f7b-2f0f-b96d98c66a5a}
   Method HomeStateMachine: Id {d40899d6-7938-037f-0dae-15b0ce72f47f}
   Method HomeTransferArm: Id {f3a5e492-51cd-0ddd-390f-6110239748db}
   Method InitHomeGarage: Id {e972dcc7-7e74-0d95-00e2-3f2f25e31bf0}
   Method InitHomeTransferArm: Id {019233af-4578-0d4f-2ca9-f60e02147d24}
   Method InitRotateGarageForClearance: Id {7e2aba46-38f3-0adf-16a6-38b66936ce8e}
   Method InitSelectGarageSlotForLoading: Id {c61e3c89-11bd-0130-00ce-6ad87d562048}
   Method InitSelectGarageSlotForRemoval: Id {f2d07db5-4e89-073a-1bd2-525077f83d27}
   Method ManualControl: Id {75581a9d-1fae-0f7c-133f-c967f378fea2}
   Method MoveToGarageSlotFaceTransferArm: Id {3cf1bab1-d70d-0336-2005-295dae3152a4}
   Method MoveToGarageSlotHeight: Id {50a35882-1804-0b08-1081-a423427c611f}
   Method RetractGarage: Id {d9daa368-9b47-09f6-01fd-88aca31ba63a}
   Method RotateGarageForClearance: Id {349e47cb-9e0e-0f8e-2b8f-84e6b8fa4669}
   Method RotateGarageForClearanceManual: Id {8a0bce26-7aa7-0334-0ae2-24e4e79d422c}
   Method RotateToFacePort: Id {a1bcadb9-002a-0cff-0d5c-dd11387aa595}
   Method RotateToFaceTransferArm: Id {8644950d-6572-0c21-1ab0-fa5ee03dc8b2}
   Method ScrewSampleIntoGarage: Id {709b251d-e374-03ca-14e4-1fe775d4a50f}
   Method SelectDesiredAction: Id {430e1a14-0c94-0a6d-0a52-e979706575e1}
   Method SelectGarageSlotForLoading: Id {2b10747f-2ffd-01ee-377b-adb0823b9413}
   Method SelectGarageSlotForRemoval: Id {eacea1be-0497-0bdd-04d8-27aa274fb735}
   Method SelectLoadUnloadGarage: Id {a35c3c83-d238-09ef-3607-5155cde28cc1}
   Method SetPositionStateWaitForArrivalQuitIfError: Id {d44e2606-d30e-0dfa-0e6d-d39d755dd87c}
   Method SetSeqState: Id {5732567c-ff6f-0fc6-00b4-ad7738497567}
   Method SetState: Id {f0976d71-98de-093b-2162-d355b7bb1b7a}
   Method SetSubstate: Id {31db8c10-c435-0cb2-3996-0d4292874597}
   Method StateMachine: Id {18b416ce-bd12-0d40-24f1-ec051178da5e}
   Method StateMachine_statechart: Id {7a069fbc-18fd-030c-07da-d834eec6f82c}
   Method UnscrewSampleFromGarage: Id {3464dcca-0819-0f26-0b96-1ede58811e89}
   Method UpdateLoadUnloadAbleStatuses: Id {e68786cd-675c-079a-1ee4-032b6bf55b9a}
   Method UpdatePositionStates: Id {5ac718fe-1224-0ef1-1133-344bf58c49d2}
   Method UpdateSampleLocationDatabaseGarageToArm: Id {e2889859-a73f-0c94-0d3c-77770598f619}
   Method UpdateSampleLocationDatabaseManualExtraction: Id {d484c4e3-0eb4-0b09-1524-19e30f3fb155}
   Method UpdateSampleLocationDatabaseManualInsertion: Id {7c97ebec-2d6c-02c9-0635-1131bb2f288f} *)
